PROGRAM MAIN
VAR
END_VAR

END_PROGRAM

(* stored: Version 1.1.0.1
   POU MAIN: Id {1756b2ac-ad29-44c4-877f-3b588324f484} *)
